// TIA Portal V17 export
// export: Created 2025-08-05T09:36:01.5275469Z, ExportSetting WithDefaults, DisplayName Totally Integrated Automation Portal, DisplayVersion V17, DisplayName TIA Portal Openness, DisplayVersion V17, DisplayName TIA Portal Version Control Interface, DisplayVersion V17, DisplayName SINAMICS Startdrive Advanced, DisplayVersion V17, DisplayName SINAMICS Startdrive G130, G150, S120, S150, SINAMICS MV, S210, DisplayVersion V17, DisplayName SINAMICS Startdrive G110M, G120, G120C, G120D, G120P, G115D, DisplayVersion V17, DisplayName STEP 7 Professional, DisplayVersion V17, DisplayName STEP 7 Safety, DisplayVersion V17, DisplayName WinCC Advanced, DisplayVersion V17
TYPE "LaserComm_Instance"
// stored: IsFailsafeCompliant false
   STRUCT
      API : Struct   // Tags associated with JLR Middleware and LDD
         Job : DInt;   // API Job - Triggers Job to Middleware. Value Clears on Completion of Job
         Faults : DInt;   // Faults Generated from SIS Interface. Set Bitwise
         Reset : Bool;   // Reset API
         Inputs : "API_Inputs";   // Inputs to API. Set from Middleware
         Outputs { S7_SetPoint := 'True'} : "API_Outputs";   // Outputs from API. Read by Middleware
         Parameters { S7_SetPoint := 'True'} : "API_Parameters";   // API Parameters
      END_STRUCT;
      Scanner : Struct   // Tags associated with IPG Scanner Software and Hardware
         oJob : Byte;   // Output Job Number to IPG Weld
         oGroup : Byte;   // Output Group Number to IPG Weld
         iJob : Byte;   // Input Running Job Number from IPG
         iGroup : Byte;   // Input Running Group Number from IPG Weld
         Faults : DInt;   // Faults Generated from IPG Interface. Set Bitwise
         Start : Bool;   // Start Command to IPG Weld to Execute Weld Job
         Waiting_Start : Bool;   // IPG Weld is Waiting for a Start Signal. Job and Group have been Loaded
         Waiting_Strobe : Bool;   // IPG Weld is Ready for a New Job and Group Load
         Reset : Bool;   // Reset IPG Weld Interface
         Weld_Offset : Struct   // Offset Values of Weld Position. Can be expanded to array. Not support at present.
            X : Real;   // X
            Y : Real;   // Y
            Z : Real;   // Z
            "A" : Real;   // A
            "B" : Real;   // B
            C : Real;   // C
         END_STRUCT;
      END_STRUCT;
      Static : Struct   // Static Tags used internally to Laser Comm FBs
         IPG_Job_Complete : Bool;   // IPG Weld Job has Completed
         LDD_Job_Loaded : Bool;   // LDD Sequence has been Loaded for the Part
         OverPen_Detected : Bool;   // LDD has Reported an Over Penetration. Flag set in FB.
      END_STRUCT;
   END_STRUCT;
END_TYPE
